{attribute 'qualified_only'}
VAR_GLOBAL
	nCounter : LREAL;
	sine : LREAL;
END_VAR

(* stored: Version 1.1.0.1, ProductVersion 3.1.4024.12
   GVL GVL: Id {752441fe-b960-45d5-bc60-2c0c93f55d57} *)
